FUNCTION_BLOCK AE_AX_TO_AE_SPLIT (* Gespiegelte Version von AE_TO_AE_AX_SPLIT (Plug/Socket 1:1 vertauscht): relays a bidirectional AE_AX Socket's incoming trigger onward as a unidirectional AE Plug (Trigger passthrough), plus an AX Socket injects an externally supplied value as the AE_AX Socket's outgoing backward (state) channel *)
  (* Standard: 61499-2; Function: Any Event received on OUT (AE_AX Socket, its incoming/E1 side) is forwarded onward unchanged via IN (AE Plug); whatever is received on AX_OUT (AX Socket) is relayed as the backward Event/Bool sent out via OUT (the AE_AX Socket's own outgoing EI1/DI1 side).; Description: Copyright (c) 2026 HR Agrartechnik GmbH This program and the accompanying materials are made available under the terms of the Eclipse Public License 2.0 which is available at https://www.eclipse.org/legal/epl-2.0/ SPDX-License-Identifier: EPL-2.0 *)
  (* Version 1.0, 2026-09-12, Franz Höpfinger, HR Agrartechnik GmbH, Initial Version - gespiegelt von AE_TO_AE_AX_SPLIT (Plug/Socket 1:1 vertauscht). *)
  PACKAGE adapter::events::bidirectional;
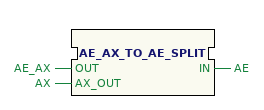
  SOCKETS
    OUT : adapter::types::bidirectional::AE_AX; (* Input (Trigger in, Zustand out) *)
    AX_OUT : adapter::types::unidirectional::AX; (* feeds the AE_AX backward (state) channel *)
  END_SOCKETS
  PLUGS
    IN : adapter::types::unidirectional::AE; (* Output (Trigger, unidirectional) *)
  END_PLUGS
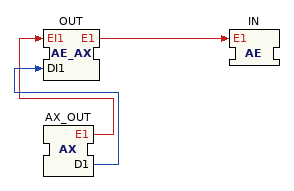
  EVENT_CONNECTIONS
    OUT.E1 TO IN.E1;
    AX_OUT.E1 TO OUT.EI1;
  END_CONNECTIONS
  DATA_CONNECTIONS
    AX_OUT.D1 TO OUT.DI1;
  END_CONNECTIONS
END_FUNCTION_BLOCK
